FUNCTION_BLOCK FB_SerialCom
VAR_IN_OUT
	TxBuffer	: ComBuffer;
	RxBuffer	: ComBuffer;
END_VAR
VAR
	Timer		: TON := (PT:=T#5S); // Timer für Sendezyklus
	fbSend		: SendString;
	bSendBusy	: BOOL;
	eSendErrorID: ComError_t;

	(* 	ReceiveString kann 80 Zeichen empfangen
		Wenn mehr Platz gebraucht: -> ReceiveString255 *)
	fbReceive		: ReceiveString;
	sReceivedString	: STRING;
	sLastReceivedString: STRING;
	bStringReceived	: BOOL;
	bReceiveBusy	: BOOL;
	bReceiveError	: BOOL;
	eReceiveErrorID	: ComError_t;
	bReceiveTimeout	: BOOL;
	nReceiveCounter	: UDINT;
END_VAR

(* fbSend wird alle x Sekunden aktiviert, um den Sendstring zu senden
   fbSend wird auch aktiviert, wenn der String nach einem Zyklus noch nicht fertig gesendet wurde
   (d.h. wenn Busy = True ist)
*)
Timer(IN:=TRUE);
IF Timer.Q OR fbSend.Busy THEN
	Timer(IN:=FALSE); (* reset timer *)
	fbSend(
			SendString:= 'Hello World! Here I am! Go Robo!!!#',  // Hier Nachricht definieren
			TXbuffer:= TxBuffer,
			Busy=> bSendBusy,
			Error=> );
	IF fbSend.Error <> COMERROR_NOERROR THEN
		eSendErrorID := fbSend.Error;
	END_IF
END_IF

(* fbReceive empfängt Daten, die mit \02 anfangen und \03 aufhören
	Prefix und Suffix können auch anders gewählt werden oder leer sein
	(leer -> fbReceive empfängt dauerhaft)
*)
fbReceive(	
	Prefix:= '$02',	// $02 == \02 ascii
	Suffix:= '$03',	// $03 == \03 ascii
	Timeout:= T#3S,
	ReceivedString:= sReceivedString, // empfangene Nachricht
	RXbuffer:= RxBuffer,
	StringReceived=> bStringReceived,
	Busy=> bReceiveBusy,
	Error=> ,
	RxTimeout=> bReceiveTimeout );
IF fbReceive.Error <> COMERROR_NOERROR THEN
	eReceiveErrorID := fbReceive.Error;
END_IF

// Counter how many messages are recieved
IF bStringReceived THEN
	nReceiveCounter := nReceiveCounter + 1;
	sLastReceivedString := sReceivedString;
END_IF

END_FUNCTION_BLOCK

(* stored: Version 1.1.0.1, ProductVersion 3.1.4022.3
   POU FB_SerialCom: Id {181e7c70-138b-446a-a6f5-34e588388885}, SpecialFunc None *)
